Staubli VAL3: Header.pjx

--- Header.pjx ---
Parameters version=s7.7.2 stackSize=5000 millimeterUnit=true
Program file=start.pgx
Program file=stop.pgx
Data file=Header.dtx

--- Header.dtx ---
mdesc mNomSpeed
public num nMsgType
public num nCommType
public num nReplyCode
